Staubli VAL3: onBackSpace.pgx

program onBackSpace(bool& x_bSave[])
  local string l_sName
  local num l_nX
  local num l_nY
  local string l_sNewName
  local string l_sMessage
  local bool l_bFound
begin
  //
  // NB sEvent is the selected
  // element in the LIST
  //
  // enter the name of the preset
  //

    call axis:get(l_sName,nIndex)
    // change the name
    if l_sName!=""
      l_nX=40-use:nBottomX+find(sEvent,l_sName)-1
      l_nY=nView+1
      // read the new name string
      l_sNewName=l_sName
      call use:read(l_nX,l_nY,l_sNewName,10,false)
      if l_sName!=l_sNewName and l_sNewName!=""
        call axis:find(l_sNewName,l_bFound)
        if l_bFound
          call language:message(l_sMessage,-2)
        else
          call axis:set(l_sNewName,nIndex)
          x_bSave=true
          call buildList()
        endIf
      endIf
    endIf

end
